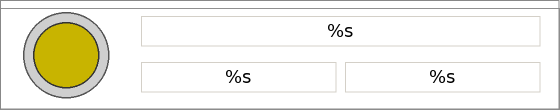
VISUALIZATION SingleSafeInput  // 560x110
VAR_IN_OUT
	stDigitalInput : ST_VisuCtrlInputFrame;
END_VAR
    GroupBox (0,0 560x110)
        Lamp1 (16,5 100x100), variable: stDigitalInput.bIn, style: Lamp-Lamp1-Yellow
        Textfield (141,16 399x30), "%s", text variable: stDigitalInput.sName
        Textfield (345,62 195x30), "%s", text variable: stDigitalInput.sPortID
        Textfield (141,62 195x30), "%s", text variable: stDigitalInput.sModuleType
END_VISUALIZATION

(* stored: Version 1.1.0.1, ProductVersion 3.1.4024.12
   Visu SingleSafeInput: Id {3d8f9c1c-7ec0-44f9-8360-6fea83a2395b} *)
